// TIA Portal V20 export
// export: Created 2026-07-20T07:26:35.3053543Z, ExportSetting WithDefaults, DisplayName Totally Integrated Automation Portal, DisplayVersion V20 Update 5, DisplayName TIA Portal Openness, DisplayVersion V20 Update 4, DisplayName TIA Portal Version Control Interface, DisplayVersion V20 Update 5, DisplayName SINAMICS Startdrive Advanced, DisplayVersion V20, DisplayName SINAMICS DCC, DisplayVersion V20, DisplayName SINAMICS Startdrive G130, G150, S120, S150, SINAMICS MV, G220, S200, S210, DisplayVersion V20, DisplayName SINAMICS Startdrive G110M, G120, G120C, G120D, G120P, G115D, DisplayVersion V20, DisplayName STEP 7 Professional, DisplayVersion V20 Update 5, DisplayName STEP 7 Safety, DisplayVersion V20 Update 2, DisplayName WinCC Basic/Comfort/Advanced, DisplayVersion V20 Update 5, DisplayName WinCC Unified, DisplayVersion V20 Update 5
FUNCTION "AnalogScale" : Void   // FC28, LAD
TITLE = Analog Scaling
{ S7_Optimized_Access := 'TRUE' }
VERSION : 0.1
// stored: AutoNumber true, IsIECCheckEnabled false, SetENOAutomatically false, UDAEnableTagReadback false
   VAR_INPUT
      Input : Real;
      Input_Min : Real;
      Input_Max : Real;
      Scaled_Min : Real;
      Scaled_Max : Real;
   END_VAR
   VAR_OUTPUT
      Output : Real;
   END_VAR
   VAR_TEMP
      InTemp : Real;
      Temp1 : Real;
      Temp2 : Real;
      Temp3 : Real;
      Temp4 : Real;
      Temp5 : Real;
   END_VAR
BEGIN

REGION Network 1
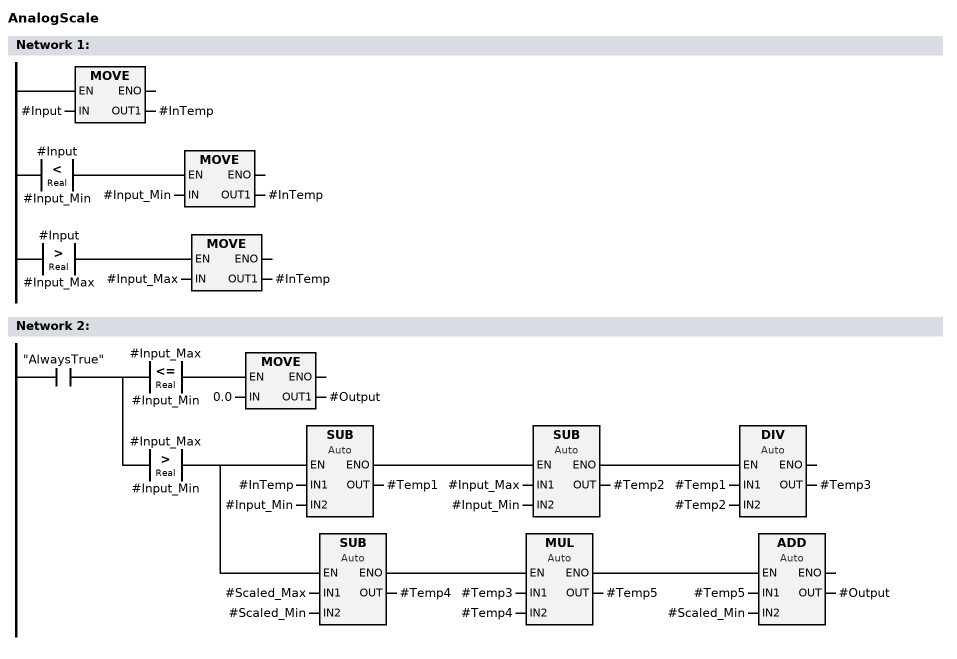
   RUNG wire#powerrail
      Move(in := #Input, out1 => #InTemp)
   END_RUNG
   RUNG wire#powerrail
      { S7_Templates := "SrcType := Real" } LT_Contact(in1 := #Input, in2 := #Input_Min)
      Move(in := #Input_Min, out1 => #InTemp)
   END_RUNG
   RUNG wire#powerrail
      { S7_Templates := "SrcType := Real" } GT_Contact(in1 := #Input, in2 := #Input_Max)
      Move(in := #Input_Max, out1 => #InTemp)
   END_RUNG
   // the same network as SCL:
   #InTemp := #Input;
   IF #Input < #Input_Min THEN #InTemp := #Input_Min; END_IF;
   IF #Input > #Input_Max THEN #InTemp := #Input_Max; END_IF;
END_REGION

REGION Network 2
   RUNG wire#powerrail
      Contact( "AlwaysTrue" )
      wire#w1
      { S7_Templates := "SrcType := Real" } LE_Contact(in1 := #Input_Max, in2 := #Input_Min)
      Move(in := 0.0, out1 => #Output)
   END_RUNG
   RUNG wire#w1
      { S7_Templates := "SrcType := Real" } GT_Contact(in1 := #Input_Max, in2 := #Input_Min)
      wire#w2
      Sub(in1 := #InTemp, in2 := #Input_Min, out => #Temp1)
      Sub(in1 := #Input_Max, in2 := #Input_Min, out => #Temp2)
      Div(in1 := #Temp1, in2 := #Temp2, out => #Temp3)
   END_RUNG
   RUNG wire#w2
      Sub(in1 := #Scaled_Max, in2 := #Scaled_Min, out => #Temp4)
      Mul(in1 := #Temp3, in2 := #Temp4, out => #Temp5)
      Add(in1 := #Temp5, in2 := #Scaled_Min, out => #Output)
   END_RUNG
   // the same network as SCL:
   IF "AlwaysTrue" AND (#Input_Max <= #Input_Min) THEN #Output := 0.0; END_IF;
   IF "AlwaysTrue" AND (#Input_Max > #Input_Min) THEN
       #Temp1 := #InTemp - #Input_Min;
       #Temp2 := #Input_Max - #Input_Min;
       #Temp3 := #Temp1 / #Temp2;
       #Temp4 := #Scaled_Max - #Scaled_Min;
       #Temp5 := #Temp3 * #Temp4;
       #Output := #Temp5 + #Scaled_Min;
   END_IF;
END_REGION
END_FUNCTION
